PROGRAM offline_main


VAR
	offline_1: offline_fb;
	offline_test: BOOL ;
	error_bit: BOOL;
	cyl_1_w_sol: BOOL;
	cyl_1_h_sol: BOOL;
	cyl_h_fb_1: BOOL;
	cyl_w_fb_1: BOOL;
END_VAR

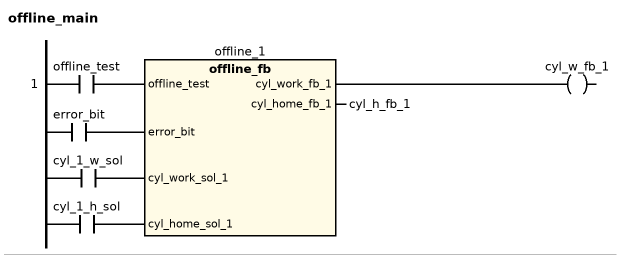
// NETWORK 1
offline_1(
    offline_test := offline_test,
    error_bit := error_bit,
    cyl_work_sol_1 := cyl_1_w_sol,
    cyl_home_sol_1 := cyl_1_h_sol,
    cyl_home_fb_1 => cyl_h_fb_1); // offline_fb
cyl_w_fb_1 := offline_1.cyl_work_fb_1;

END_PROGRAM

(* stored: Version 1.1.0.1, ProductVersion 3.1.4024.11
   POU offline_main: Id {03973bd6-d3cb-485e-a7a7-f24d52dd5fb5}, SpecialFunc None *)
